// TwinCAT 3 PLC project bts_vac
// ProgramVersion: 3.1.4023.0
// libraries:
//   Tc2_Standard, * (Beckhoff Automation GmbH)
//   Tc2_System, * (Beckhoff Automation GmbH)
//   Tc2_Utilities, * (Beckhoff Automation GmbH)
//   Tc3_Module, * (Beckhoff Automation GmbH)
//   LCLS General,2.4.2,SLAC
//   LCLS Vacuum,1.4.0,SLAC - LCLS
//   LCLSVacuumSerialDriverLib,1.2.2,SLAC - LCLS
//   PMPS,0.15.3,SLAC - LCLS
// project tree:
//   DUTs/ E_TransportTube.TcDUT (not stored), ST_TransportTubeConfig.TcDUT (not stored), ST_TransportTubeDevices.TcDUT (not stored), T_TransportTube.TcDUT (not stored)
//   DUTs/Operations/ E_Op.TcDUT (not stored), E_OpStep.TcDUT (not stored)
//   DUTs/SystemStatusChecks/ E_GaugeCompOp.TcDUT (not stored)
//   DUTs/SystemStatusChecks/Switchbox/ ST_SBGaugeReadings.TcDUT, ST_SBGaugeReadingsOp.TcDUT, ST_SBPumpStatuses.TcDUT (not stored), ST_SBValveStatuses.TcDUT (not stored)
//   DUTs/SystemStatusChecks/TransportTubes/ ST_TransportTubeOps.TcDUT (not stored), ST_TransportTubeStatuses.TcDUT (not stored)
//   GVLs/ GVL_BTS_VAC.TcGVL, GVL_Constants.TcGVL (not stored), GVL_MaintainLaser.TcGVL (not stored), GVL_Operation.TcGVL (not stored), GVL_TransportTubes.TcGVL (not stored)
//   / PlcTask.TcTTO (not stored)
//   POUs/ FB_TransportTube.TcPOU (not stored), F_UpdateIO.TcPOU (not stored), MAIN.TcPOU, MaintainLaser.TcPOU (not stored), Operate.TcPOU (not stored)
//   POUs/Helpers/ F_Atm.TcPOU (not stored), F_GetTransportTube.TcPOU (not stored), F_PumpStationTurboPumpInterlock.TcPOU (not stored), F_SBVentInterlock.TcPOU (not stored)
//   POUs/Operations/Abstracts/ FB_MaintainLaserOperation.TcPOU (not stored), FB_Operation.TcPOU (not stored), FB_TTOperation.TcPOU (not stored)
//   POUs/Operations/ FB_LaserOn.TcPOU (not stored), FB_OpenTransportTube.TcPOU (not stored), FB_SlowPumpSwitchbox.TcPOU (not stored), FB_SlowVentSwitchbox.TcPOU (not stored), FB_VentTransportTube.TcPOU (not stored), FB_VentPumpStation.TcPOU (not stored), FB_PumpSwitchbox.TcPOU (not stored), FB_VentSwitchbox.TcPOU, FB_PumpTransportTube.TcPOU (not stored)
//   POUs/Operations/MaintainLaser/ FB_SwitchboxIonPumpFailure.TcPOU (not stored), FB_SwitchboxRoughingOrTurboPumpFailure.TcPOU (not stored)
//   POUs/SystemStatusChecks/ F_CompareGauge.TcPOU (not stored)
//   POUs/SystemStatusChecks/Switchbox/ F_GetSBGaugeReadings.TcPOU (not stored), F_GetSBPumpStatuses.TcPOU (not stored), F_GetSBValveStatuses.TcPOU (not stored), F_SetSBPumpStatuses.TcPOU (not stored), F_SetSBValveStatuses.TcPOU, F_VerifySBGaugeReadings.TcPOU (not stored), F_VerifySBPumpStatuses.TcPOU (not stored), F_VerifySBValveStatuses.TcPOU (not stored)
//   POUs/SystemStatusChecks/TransportTubes/ F_GetTransportTubeStatuses.TcPOU (not stored), F_SetTransportTubeStatuses.TcPOU (not stored), F_VerifyAllTransportTubeStatuses.TcPOU (not stored), F_VerifyTransportTubeStatuses.TcPOU (not stored)

// ---- DUTs/SystemStatusChecks/Switchbox/ST_SBGaugeReadings.TcDUT
(* Statuses of the gauges for the switchbox *)
TYPE ST_SBGaugeReadings :
STRUCT
	(* Gauge readings *)
	
	fDPPiraniVal : REAL; // LXLHN:GPI:03
	eDPPiraniState : E_PressureState;
	
	fDPColdCathodeVal : REAL; // LXLHN:GCC:02
	eDPColdCathodeState : E_PressureState;
	
	fPumpStationPirani1Val : REAL; // LXLHN:GPI:01
	ePumpStationPirani1State : E_PressureState;
	
	fPumpStationPirani2Val : REAL; // LXLHN:GPI:02
	ePumpStationPirani2State : E_PressureState;
	
	fPumpStationColdCathodeVal : REAL; // LXLHN:GCC:01
	ePumpStationColdCathodeState : E_PressureState;
END_STRUCT
END_TYPE

// ---- DUTs/SystemStatusChecks/Switchbox/ST_SBGaugeReadingsOp.TcDUT
(* What operations should be used to compare gauge status *)
TYPE ST_SBGaugeReadingsOp :
STRUCT
	eDPPiraniOp : E_GaugeCompOp; // LXLHN:GPI:03
	eDPColdCathodeOp : E_GaugeCompOp; // LXLHN:GCC:02
	ePumpStationPirani1Op : E_GaugeCompOp; // LXLHN:GPI:01
	ePumpStationPirani2Op : E_GaugeCompOp; // LXLHN:GPI:02
	ePumpStationColdCathodeOp : E_GaugeCompOp; // LXLHN:GCC:01
END_STRUCT
END_TYPE

// ---- GVLs/GVL_BTS_VAC.TcGVL
{attribute 'qualified_only'}
VAR_GLOBAL
	(* Valves *)	
	fb_PP_VGC_FFOut : FB_HardwareFFOutput;
	
	{attribute 'pytmc'	  :=	' pv: LXLHN:VGC:01 '}
	{attribute 'TcLinkTo' := 	'.i_xOpnLS			:=	TIIB[EL1004_02_12]^Channel 2^Input;
								 .i_xClsLS			:=	TIIB[EL1004_02_12]^Channel 1^Input;
								 .q_xOPN_DO			:=	TIIB[EL2004_02_14]^Channel 2^Output'}
	fb_PP_VGC : FB_VGC; // Gate valve, vacuum switchbox
	
	{attribute 'pytmc' 	  :=	' pv: LXLHN:VVC:01 '}
	{attribute 'TcLinkTo' := 	'.q_xOPN_DO			:=	TIIB[EL2004_02_05]^Channel 3^Output'}
	fb_PP_VVC : FB_VVC; // Turbo N2 purge
	
	
	{attribute 'pytmc'	  :=	' pv: LXLHN:VRC:01 '}
	{attribute 'TcLinkTo' := 	'.i_xOpnLS			:=	TIIB[EL1002_02_01]^Channel 2^Input;
								 .i_xClsLS			:=	TIIB[EL1002_02_01]^Channel 1^Input;
								 .q_xOPN_DO			:=	TIIB[EL2004_02_04]^Channel 1^Output'}
	fb_PP_VRC_1 : FB_VRC; // O-ring diff pump valve
	
	{attribute 'pytmc'	  :=	' pv: LXLHN:VRC:02 '}
	{attribute 'TcLinkTo' := 	'.i_xOpnLS			:=	TIIB[EL1002_02_02]^Channel 2^Input;
								 .i_xClsLS			:=	TIIB[EL1002_02_02]^Channel 1^Input;
								 .q_xOPN_DO			:=	TIIB[EL2004_02_04]^Channel 3^Output'}
	fb_PP_VRC_2 : FB_VRC; // Foreline valve
	
	{attribute 'pytmc'	  :=	' pv: LXLHN:VRC:03 '}
	{attribute 'TcLinkTo' := 	'.i_xOpnLS			:=	TIIB[EL1002_02_03]^Channel 2^Input;
								 .i_xClsLS			:=	TIIB[EL1002_02_03]^Channel 1^Input;
								 .q_xOPN_DO			:=	TIIB[EL2004_02_04]^Channel 4^Output'}
	fb_PP_VRC_3 : FB_VRC; // Slow pump valve
	
	st_VP_VVC_1 : ST_VCC_NO;
	{attribute 'pytmc' 	  :=	' pv: LXLHN:VVC:02 '}
	{attribute 'TcLinkTo' := 	'.q_xOPN_DO			:=	TIIB[EL2004_02_05]^Channel 1^Output'}
	fb_VP_VVC_1 : FB_VCC_NO; // Vent valve, Switchbox
	
	st_VP_VVC_2 : ST_VCC_NO;
	{attribute 'pytmc' 	  :=	' pv: LXLHN:VVC:032 '}
	{attribute 'TcLinkTo' := 	'.q_xOPN_DO			:=	TIIB[EL2004_02_05]^Channel 2^Output'}
	fb_VP_VVC_2 : FB_VCC_NO; // Vent valve, Slow, Switchbox

	
	(* Pumps *)
	{attribute 'pytmc' 	  := ' 	
		pv: LXLHN:PTM:01
		io: io 
	'}
	{attribute 'TcLinkTo' := 	'.i_xAtSpd			:=	TIIB[EL1004_00_03]^Channel 3^Input;
								 .i_xRemote			:=	TIIB[EL1004_00_03]^Channel 2^Input;
								 .i_xFaultNC		:=	TIIB[EL1004_00_03]^Channel 1^Output;
								 .q_RunDO			:=	TIIB[EL2004_00_04]^Channel 1^Input;
								 .q_xRemote			:=	TIIB[EL2004_00_04]^Channel 2^Input;								 
								 .q_PumpingStation	:=	TIIB[EL2004_00_04]^Channel 3^Output;'}								
	fb_PP_PTM : FB_PTM_Pfeiffer; // Turbo pump
	
	{attribute 'pytmc' 	  := ' 	
		pv: LXLHN:PMF:01
		io: io 
	'}
	{attribute 'TcLinkTo' := 	'.i_xWarning		:=	TIIB[EL1004_00_01]^Channel 4^Input;
								 .i_xAlarm			:=	TIIB[EL1004_00_01]^Channel 3^Input;
								 .i_xLocal			:=	TIIB[EL1004_00_01]^Channel 2^Output;
								 .i_xIsRun			:=	TIIB[EL1004_00_01]^Channel 1^Output;								 
								 .q_xRunDO			:=	TIIB[EL2794_00_02]^Channel 1^Input;
								 .q_xLspdDO			:=	TIIB[EL2794_00_02]^Channel 2^Input;								 
								 .q_xResetDo		:=	TIIB[EL2794_00_02]^Channel 3^Output;'}	
	fb_PP_PMF : FB_KashiyamaPump; // Roughing Pump
	
	{attribute 'pytmc'    := 	' pv: LXLHN:PP:PIP'}
	{attribute 'TcLinkTo' := 	'.i_iPRESS			:=	TIIB[EL3064_00_08]^AI Standard Channel 3^Value;
								 .i_xSP_DI			:= 	TIIB[EL1004_00_07]^Channel 3^Input;
								 .q_xHVEna_DO		:= 	TIIB[EL2794_00_06]^Channel 3^Output'}
	fb_PP_PIP : FB_PIP_Gamma; // Ion Pump, SW
	
	(* Gauges *)
	{attribute 'pytmc' 	  :=	' pv: LXLHN:GPI:01 '}
	{attribute 'TcLinkTo' := 	'.i_iPRESS_R		:=	TIIB[EL3174_01_10]^AI Standard Channel 3^Value '}
	fb_PP_GPI_1 : FB_MKS275; // Switchbox pumpline ATM gauge
	
	{attribute 'pytmc' 	  :=	' pv: LXLHN:GPI:02 '}
	{attribute 'TcLinkTo' := 	'.i_iPRESS_R		:=	TIIB[EL3174_01_11]^AI Standard Channel 1^Value '}
	fb_PP_GPI_2 : FB_MKS275; // Foreline gauge
	
	{attribute 'pytmc' 	  :=	' pv: LXLHN:GPI:03 '}
	{attribute 'TcLinkTo' := 	'.i_iPRESS_R		:=	TIIB[EL3174_01_10]^AI Standard Channel 2^Value '}
	fb_DP_GPI : FB_MKS275; // Switchbox gauge
	
	{attribute 'pytmc' 	  :=	' pv: LXLHN:GCC:01 '}
	{attribute 'TcLinkTo' := 	'.i_iPRESS_R		:=	TIIB[EL3174_01_09]^AI Standard Channel 2^Value;
								 .i_xHV_ON	    	:=	TIIB[EL1124_01_06]^Channel 1^Input;
								 .i_xDisc_Active	:=	TIIB[EL1124_01_06]^Channel 2^Input;
								 .q_xHV_DIS			:= 	TIIB[EL2624_01_02]^Channel 2^Output	'}
	fb_PP_GCC : FB_MKS500; // Switchbox pumpline Cold Cathode gauge
	
	{attribute 'pytmc' 	  :=	' pv: LXLHN:GCC:02 '}
	{attribute 'TcLinkTo' := 	'.i_iPRESS_R		:=	TIIB[EL3174_01_09]^AI Standard Channel 4^Value;
								 .i_xHV_ON	    	:=	TIIB[EL1124_01_07]^Channel 3^Input;
								 .i_xDisc_Active	:=	TIIB[EL1124_01_07]^Channel 4^Input;
								 .q_xHV_DIS			:= 	TIIB[EL2624_01_02]^Channel 4^Output	'}
	fb_DP_GCC : FB_MKS500; // Switchbox Cold Cathode gauge
	
	(* Transport Tubes *)
	// LS1
	fb_LS1_VGC_FFOut : FB_HardwareFFOutput;
	{attribute 'pytmc'	  :=	' pv: LTLHN:LS1:VGC:01 '}
	{attribute 'TcLinkTo' := 	'.i_xOpnLS			:=	TIIB[EL1004_02_06]^Channel 2^Input;
								 .i_xClsLS			:=	TIIB[EL1004_02_06]^Channel 1^Input;
								 .q_xOPN_DO			:=	TIIB[EL2004_02_08]^Channel 1^Output'}
	fb_LS1_VGC : FB_VGC; // Gate valve, Input LS1 laser Table
	{attribute 'pytmc'    := 	' pv: LTLHN:LS1:PIP:01 '}
	{attribute 'TcLinkTo' := 	'.i_iPRESS			:=	TIIB[EL3064_00_08]^AI Standard Channel 2^Value;
								 .i_xSP_DI			:= 	TIIB[EL1004_00_07]^Channel 2^Input;
								 .q_xHVEna_DO		:= 	TIIB[EL2794_00_06]^Channel 2^Output'}
	fb_LS1_PIP : FB_PIP_Gamma; // Ion Pump, input tube LS1
	{attribute 'pytmc' 	  :=	' pv: LTLHN:LS1:GPI:01 '}
	{attribute 'TcLinkTo' := 	'.i_iPRESS_R		:=	TIIB[EL3174_01_10]^AI Standard Channel 4^Value '}
	fb_LS1_GPI : FB_MKS275; // Input tube LS1 ATM gauge
	{attribute 'pytmc' 	  :=	' pv: LTLHN:LS1:GCC:01 '}
	{attribute 'TcLinkTo' := 	'.i_iPRESS_R		:=	TIIB[EL3174_01_09]^AI Standard Channel 3^Value;
								 .i_xHV_ON	    	:=	TIIB[EL1124_01_06]^Channel 3^Input;
								 .i_xDisc_Active	:=	TIIB[EL1124_01_06]^Channel 4^Input;
								 .q_xHV_DIS			:= 	TIIB[EL2624_01_02]^Channel 3^Output	'}
	fb_LS1_GCC : FB_MKS500; // Input tube LS1, Cold Cathode gauge
	
	// LS5
	fb_LS5_VGC_FFOut : FB_HardwareFFOutput;
	{attribute 'pytmc'	  :=	' pv: LTLHN:LS5:VGC:01 '}
	{attribute 'TcLinkTo' := 	'.i_xOpnLS			:=	TIIB[EL1004_02_09]^Channel 4^Input;
								 .i_xClsLS			:=	TIIB[EL1004_02_09]^Channel 3^Input;
								 .q_xOPN_DO			:=	TIIB[EL2004_02_11]^Channel 2^Output'}
	fb_LS5_VGC : FB_VGC; // Gate valve, Input LS5 laser Table
	{attribute 'pytmc'    := 	' pv: LTLHN:LS5:PIP:01 '}
	{attribute 'TcLinkTo' := 	'.i_iPRESS			:=	TIIB[EL3064_00_11]^AI Standard Channel 4^Value;
								 .i_xSP_DI			:= 	TIIB[EL1004_00_10]^Channel 4^Input;
								 .q_xHVEna_DO		:= 	TIIB[EL2794_00_09]^Channel 4^Output'}
	fb_LS5_PIP : FB_PIP_Gamma; // Ion Pump, input tube LS5
	{attribute 'pytmc' 	  :=	' pv: LTLHN:LS5:GPI:01 '}
	{attribute 'TcLinkTo' := 	'.i_iPRESS_R		:=	TIIB[EL3174_03_13]^AI Standard Channel 1^Value '}
	fb_LS5_GPI : FB_MKS275; // Input tube LS5 ATM gauge
	{attribute 'pytmc' 	  :=	' pv: LTLHN:LS5:GCC:01 '}
	{attribute 'TcLinkTo' := 	'.i_iPRESS_R		:=	TIIB[EL3174_03_11]^AI Standard Channel 1^Value;
								 .i_xHV_ON	    	:=	TIIB[EL1124_03_08]^Channel 1^Input;
								 .i_xDisc_Active	:=	TIIB[EL1124_03_08]^Channel 2^Input;
								 .q_xHV_DIS			:= 	TIIB[EL2624_03_02]^Channel 1^Output	'}
	fb_LS5_GCC : FB_MKS500; // Input tube LS5, Cold Cathode gauge
	
	// LS8
	fb_LS8_VGC_FFOut : FB_HardwareFFOutput;
	{attribute 'pytmc'	  :=	' pv: LTLHN:LS8:VGC:01 '}
	{attribute 'TcLinkTo' := 	'.i_xOpnLS			:=	TIIB[EL1004_02_09]^Channel 2^Input;
								 .i_xClsLS			:=	TIIB[EL1004_02_09]^Channel 1^Input;
								 .q_xOPN_DO			:=	TIIB[EL2004_02_11]^Channel 3^Output'}
	fb_LS8_VGC : FB_VGC; // Gate valve, Input LS8 laser Table
	{attribute 'pytmc'    := 	' pv: LTLHN:LS8:PIP:01 '}
	{attribute 'TcLinkTo' := 	'.i_iPRESS			:=	TIIB[EL3064_00_11]^AI Standard Channel 3^Value;
								 .i_xSP_DI			:= 	TIIB[EL1004_00_10]^Channel 3^Input;
								 .q_xHVEna_DO		:= 	TIIB[EL2794_00_09]^Channel 3^Output'}
	fb_LS8_PIP : FB_PIP_Gamma; // Ion Pump, input tube LS8
	{attribute 'pytmc' 	  :=	' pv: LTLHN:LS8:GPI:01 '}
	{attribute 'TcLinkTo' := 	'.i_iPRESS_R		:=	TIIB[EL3174_03_13]^AI Standard Channel 2^Value '}
	fb_LS8_GPI : FB_MKS275; // Input tube LS8 ATM gauge
	{attribute 'pytmc' 	  :=	' pv: LTLHN:LS8:GCC:01 '}
	{attribute 'TcLinkTo' := 	'.i_iPRESS_R		:=	TIIB[EL3174_03_11]^AI Standard Channel 2^Value;
								 .i_xHV_ON	    	:=	TIIB[EL1124_03_08]^Channel 3^Input;
								 .i_xDisc_Active	:=	TIIB[EL1124_03_08]^Channel 4^Input;
								 .q_xHV_DIS			:= 	TIIB[EL2624_03_02]^Channel 2^Output	'}
	fb_LS8_GCC : FB_MKS500; // Input tube LS8, Cold Cathode gauge

	// LD2
	fb_LD2_VGC_FFOut : FB_HardwareFFOutput;
	{attribute 'pytmc'	  :=	' pv: LTLHN:LD2:VGC:01 '}
	{attribute 'TcLinkTo' := 	'.i_xOpnLS			:=	TIIB[EL1004_02_12]^Channel 4^Input;
								 .i_xClsLS			:=	TIIB[EL1004_02_12]^Channel 3^Input;
								 .q_xOPN_DO			:=	TIIB[EL2004_02_14]^Channel 3^Output'}
	fb_LD2_VGC : FB_VGC; // Gate valve, Output tube LD2 laser Table
	{attribute 'pytmc'    := 	' pv: LTLHN:LD2:PIP:01 '}
	{attribute 'TcLinkTo' := 	'.i_iPRESS			:=	TIIB[EL3064_00_08]^AI Standard Channel 1^Value;
								 .i_xSP_DI			:= 	TIIB[EL1004_00_07]^Channel 1^Input;
								 .q_xHVEna_DO		:= 	TIIB[EL2794_00_06]^Channel 1^Output'}
	fb_LD2_PIP : FB_PIP_Gamma; // Ion Pump, output tube LD2
	{attribute 'pytmc' 	  :=	' pv: LTLHN:LD2:GPI:01 '}
	{attribute 'TcLinkTo' := 	'.i_iPRESS_R		:=	TIIB[EL3174_01_10]^AI Standard Channel 1^Value '}
	fb_LD2_GPI : FB_MKS275; // Output tube LD2 ATM gauge
	{attribute 'pytmc' 	  :=	' pv: LTLHN:LD2:GCC:01 '}
	{attribute 'TcLinkTo' := 	'.i_iPRESS_R		:=	TIIB[EL3174_01_09]^AI Standard Channel 1^Value;
								 .i_xHV_ON	    	:=	TIIB[EL1124_01_07]^Channel 1^Input;
								 .i_xDisc_Active	:=	TIIB[EL1124_01_07]^Channel 2^Input;
								 .q_xHV_DIS			:= 	TIIB[EL2624_01_02]^Channel 1^Output	'}
	fb_LD2_GCC : FB_MKS500; // Output tube LD2, Cold Cathode gauge
	
	// LD4
	fb_LD4_VGC_FFOut : FB_HardwareFFOutput;
	{attribute 'pytmc'	  :=	' pv: LTLHN:LD4:VGC:01 '}
	{attribute 'TcLinkTo' := 	'.i_xOpnLS			:=	TIIB[EL1004_02_10]^Channel 2^Input;
								 .i_xClsLS			:=	TIIB[EL1004_02_10]^Channel 1^Input;
								 .q_xOPN_DO			:=	TIIB[EL2004_02_11]^Channel 1^Output'}
	fb_LD4_VGC : FB_VGC; // Gate valve, Output tube LD4 laser Table
	{attribute 'pytmc'    := 	' pv: LTLHN:LD4:PIP:01 '}
	{attribute 'TcLinkTo' := 	'.i_iPRESS			:=	TIIB[EL3064_00_11]^AI Standard Channel 1^Value;
								 .i_xSP_DI			:= 	TIIB[EL1004_00_10]^Channel 1^Input;
								 .q_xHVEna_DO		:= 	TIIB[EL2794_00_09]^Channel 1^Output'}
	fb_LD4_PIP : FB_PIP_Gamma; // Ion Pump, output tube LD4
	{attribute 'pytmc' 	  :=	' pv: LTLHN:LD4:GPI:01 '}
	{attribute 'TcLinkTo' := 	'.i_iPRESS_R		:=	TIIB[EL3174_03_13]^AI Standard Channel 4^Value '}
	fb_LD4_GPI : FB_MKS275; // Output tube LD4 ATM gauge
	{attribute 'pytmc' 	  :=	' pv: LTLHN:LD4:GCC:01 '}
	{attribute 'TcLinkTo' := 	'.i_iPRESS_R		:=	TIIB[EL3174_03_11]^AI Standard Channel 4^Value;
								 .i_xHV_ON	    	:=	TIIB[EL1124_03_09]^Channel 3^Input;
								 .i_xDisc_Active	:=	TIIB[EL1124_03_09]^Channel 4^Input;
								 .q_xHV_DIS			:= 	TIIB[EL2624_03_02]^Channel 4^Output	'}
	fb_LD4_GCC : FB_MKS500; // Output tube LD4, Cold Cathode gauge
	
	// LD6
	fb_LD6_VGC_FFOut : FB_HardwareFFOutput;
	{attribute 'pytmc'	  :=	' pv: LTLHN:LD6:VGC:01 '}
	{attribute 'TcLinkTo' := 	'.i_xOpnLS			:=	TIIB[EL1004_02_13]^Channel 4^Input;
								 .i_xClsLS			:=	TIIB[EL1004_02_13]^Channel 3^Input;
								 .q_xOPN_DO			:=	TIIB[EL2004_02_14]^Channel 4^Output'}
	fb_LD6_VGC : FB_VGC; // Gate valve, Output tube LD6 laser Table
	{attribute 'pytmc'    := 	' pv: LTLHN:LD6:PIP:01 '}
	{attribute 'TcLinkTo' := 	'.i_iPRESS			:=	TIIB[EL3064_00_11]^AI Standard Channel 2^Value;
								 .i_xSP_DI			:= 	TIIB[EL1004_00_10]^Channel 2^Input;
								 .q_xHVEna_DO		:= 	TIIB[EL2794_00_09]^Channel 2^Output'}
	fb_LD6_PIP : FB_PIP_Gamma; // Ion Pump, output tube LD6
	{attribute 'pytmc' 	  :=	' pv: LTLHN:LD6:GPI:01 '}
	{attribute 'TcLinkTo' := 	'.i_iPRESS_R		:=	TIIB[EL3174_03_13]^AI Standard Channel 3^Value '}
	fb_LD6_GPI : FB_MKS275; // Output tube LD6 ATM gauge
	{attribute 'pytmc' 	  :=	' pv: LTLHN:LD6:GCC:01 '}
	{attribute 'TcLinkTo' := 	'.i_iPRESS_R		:=	TIIB[EL3174_03_11]^AI Standard Channel 3^Value;
								 .i_xHV_ON	    	:=	TIIB[EL1124_03_09]^Channel 1^Input;
								 .i_xDisc_Active	:=	TIIB[EL1124_03_09]^Channel 2^Input;
								 .q_xHV_DIS			:= 	TIIB[EL2624_03_02]^Channel 3^Output	'}
	fb_LD6_GCC : FB_MKS500; // Output tube LD6, Cold Cathode gauge

	// LD8
	fb_LD8_VGC_FFOut : FB_HardwareFFOutput;
	{attribute 'pytmc'	  :=	' pv: LTLHN:LD8:VGC:01 '}
	{attribute 'TcLinkTo' := 	'.i_xOpnLS			:=	TIIB[EL1004_02_07]^Channel 4^Input;
								 .i_xClsLS			:=	TIIB[EL1004_02_07]^Channel 3^Input;
								 .q_xOPN_DO			:=	TIIB[EL2004_02_07]^Channel 4^Output'}
	fb_LD8_VGC : FB_VGC; // Gate valve, Output tube LD8 laser Table
	{attribute 'pytmc'    := 	' pv: LTLHN:LD8:PIP:01 '}
	{attribute 'TcLinkTo' := 	'.i_iPRESS			:=	TIIB[EL3064_00_08]^AI Standard Channel 4^Value;
								 .i_xSP_DI			:= 	TIIB[EL1004_00_07]^Channel 4^Input;
								 .q_xHVEna_DO		:= 	TIIB[EL2794_00_06]^Channel 4^Output'}
	fb_LD8_PIP : FB_PIP_Gamma; // Ion Pump, output tube LD8
	{attribute 'pytmc' 	  :=	' pv: LTLHN:LD8:GPI:01 '}
	{attribute 'TcLinkTo' := 	'.i_iPRESS_R		:=	TIIB[EL3174_01_11]^AI Standard Channel 2^Value '}
	fb_LD8_GPI : FB_MKS275; // Output tube LD8 ATM gauge
	{attribute 'pytmc' 	  :=	' pv: LTLHN:LD8:GCC:01 '}
	{attribute 'TcLinkTo' := 	'.i_iPRESS_R		:=	TIIB[EL3174_01_11]^AI Standard Channel 3^Value;
								 .i_xHV_ON	    	:=	TIIB[EL1124_01_08]^Channel 1^Input;
								 .i_xDisc_Active	:=	TIIB[EL1124_01_08]^Channel 2^Input;
								 .q_xHV_DIS			:= 	TIIB[EL2624_01_01]^Channel 4^Output	'}
	fb_LD8_GCC : FB_MKS500; // Output tube LD8, Cold Cathode gauge
	
	// LD9
	fb_LD9_VGC_FFOut : FB_HardwareFFOutput;
	{attribute 'pytmc'	  :=	' pv: LTLHN:LD9:VGC:01 '}
	{attribute 'TcLinkTo' := 	'.i_xOpnLS			:=	TIIB[EL1004_02_06]^Channel 4^Input;
								 .i_xClsLS			:=	TIIB[EL1004_02_06]^Channel 3^Input;
								 .q_xOPN_DO			:=	TIIB[EL2004_02_08]^Channel 2^Output'}
	fb_LD9_VGC : FB_VGC; // Gate valve, Output tube LD9 laser Table
	{attribute 'pytmc'    := 	' pv: LTLHN:LD9:PIP:01 '}
	{attribute 'TcLinkTo' := 	'.i_iPRESS			:=	TIIB[EL3064_00_14]^AI Standard Channel 2^Value;
								 .i_xSP_DI			:= 	TIIB[EL1004_00_13]^Channel 2^Input;
								 .q_xHVEna_DO		:= 	TIIB[EL2794_00_12]^Channel 2^Output'}
	fb_LD9_PIP : FB_PIP_Gamma; // Ion Pump, output tube LD9
	{attribute 'pytmc' 	  :=	' pv: LTLHN:LD9:GPI:01 '}
	{attribute 'TcLinkTo' := 	'.i_iPRESS_R		:=	TIIB[EL3174_03_12]^AI Standard Channel 1^Value '}
	fb_LD9_GPI : FB_MKS275; // Output tube LD9 ATM gauge
	{attribute 'pytmc' 	  :=	' pv: LTLHN:LD9:GCC:01 '}
	{attribute 'TcLinkTo' := 	'.i_iPRESS_R		:=	TIIB[EL3174_03_10]^AI Standard Channel 1^Value;
								 .i_xHV_ON	    	:=	TIIB[EL1124_03_06]^Channel 1^Input;
								 .i_xDisc_Active	:=	TIIB[EL1124_03_06]^Channel 2^Input;
								 .q_xHV_DIS			:= 	TIIB[EL2624_03_01]^Channel 1^Output	'}
	fb_LD9_GCC : FB_MKS500; // Output tube LD9, Cold Cathode gauge

	// LD10
	fb_LD10_VGC_FFOut : FB_HardwareFFOutput;
	{attribute 'pytmc'	  :=	' pv: LTLHN:LD10:VGC:01 '}
	{attribute 'TcLinkTo' := 	'.i_xOpnLS			:=	TIIB[EL1004_02_07]^Channel 2^Input;
								 .i_xClsLS			:=	TIIB[EL1004_02_07]^Channel 1^Input;
								 .q_xOPN_DO			:=	TIIB[EL2004_02_07]^Channel 3^Output'}
	fb_LD10_VGC : FB_VGC; // Gate valve, Output tube LD10 laser Table
	{attribute 'pytmc'    := 	' pv: LTLHN:LD10:PIP:01 '}
	{attribute 'TcLinkTo' := 	'.i_iPRESS			:=	TIIB[EL3064_00_14]^AI Standard Channel 1^Value;
								 .i_xSP_DI			:= 	TIIB[EL1004_00_13]^Channel 1^Input;
								 .q_xHVEna_DO		:= 	TIIB[EL2794_00_12]^Channel 1^Output'}
	fb_LD10_PIP : FB_PIP_Gamma; // Ion Pump, output tube LD10
	{attribute 'pytmc' 	  :=	' pv: LTLHN:LD10:GPI:01 '}
	{attribute 'TcLinkTo' := 	'.i_iPRESS_R		:=	TIIB[EL3174_03_12]^AI Standard Channel 2^Value '}
	fb_LD10_GPI : FB_MKS275; // Output tube LD10 ATM gauge
	{attribute 'pytmc' 	  :=	' pv: LTLHN:LD10:GCC:01 '}
	{attribute 'TcLinkTo' := 	'.i_iPRESS_R		:=	TIIB[EL3174_03_10]^AI Standard Channel 2^Value;
								 .i_xHV_ON	    	:=	TIIB[EL1124_03_07]^Channel 3^Input;
								 .i_xDisc_Active	:=	TIIB[EL1124_03_07]^Channel 4^Input;
								 .q_xHV_DIS			:= 	TIIB[EL2624_03_01]^Channel 2^Output	'}
	fb_LD10_GCC : FB_MKS500; // Output tube LD10, Cold Cathode gauge	
	
	// LD14
	fb_LD14_VGC_FFOut : FB_HardwareFFOutput;
	{attribute 'pytmc'	  :=	' pv: LTLHN:LD14:VGC:01 '}
	{attribute 'TcLinkTo' := 	'.i_xOpnLS			:=	TIIB[EL1004_02_10]^Channel 4^Input;
								 .i_xClsLS			:=	TIIB[EL1004_02_10]^Channel 3^Input;
								 .q_xOPN_DO			:=	TIIB[EL2004_02_11]^Channel 4^Output'}
	fb_LD14_VGC : FB_VGC; // Gate valve, Output tube LD14 laser Table
	{attribute 'pytmc'    := 	' pv: LTLHN:LD14:PIP:01 '}
	{attribute 'TcLinkTo' := 	'.i_iPRESS			:=	TIIB[EL3064_00_14]^AI Standard Channel 3^Value;
								 .i_xSP_DI			:= 	TIIB[EL1004_00_13]^Channel 3^Input;
								 .q_xHVEna_DO		:= 	TIIB[EL2794_00_12]^Channel 3^Output'}
	fb_LD14_PIP : FB_PIP_Gamma; // Ion Pump, output tube LD14
	{attribute 'pytmc' 	  :=	' pv: LTLHN:LD14:GPI:01 '}
	{attribute 'TcLinkTo' := 	'.i_iPRESS_R		:=	TIIB[EL3174_03_12]^AI Standard Channel 3^Value '}
	fb_LD14_GPI : FB_MKS275; // Output tube LD14 ATM gauge
	{attribute 'pytmc' 	  :=	' pv: LTLHN:LD14:GCC:01 '}
	{attribute 'TcLinkTo' := 	'.i_iPRESS_R		:=	TIIB[EL3174_03_10]^AI Standard Channel 3^Value;
								 .i_xHV_ON	    	:=	TIIB[EL1124_03_07]^Channel 1^Input;
								 .i_xDisc_Active	:=	TIIB[EL1124_03_07]^Channel 2^Input;
								 .q_xHV_DIS			:= 	TIIB[EL2624_03_01]^Channel 3^Output	'}
	fb_LD14_GCC : FB_MKS500; // Output tube LD14, Cold Cathode gauge

END_VAR

// ---- POUs/MAIN.TcPOU
PROGRAM MAIN
VAR
END_VAR

(* Update physical IO signals *)
F_UpdateIO();

(* Update transport tubes *)
GVL_TransportTubes.fbLS1(
	i_stConfig := GVL_TransportTubes.stLS1, 
	i_bLaserExtIntl := TRUE
);

GVL_TransportTubes.fbLS5(
	i_stConfig := GVL_TransportTubes.stLS5, 
	i_bLaserExtIntl := TRUE
);

GVL_TransportTubes.fbLS8(
	i_stConfig := GVL_TransportTubes.stLS8, 
	i_bLaserExtIntl := TRUE
);

GVL_TransportTubes.fbLD2(
	i_stConfig := GVL_TransportTubes.stLD2,
	i_bLaserExtIntl := TRUE
);

GVL_TransportTubes.fbLD4(
	i_stConfig := GVL_TransportTubes.stLD4,
	i_bLaserExtIntl := TRUE
);

GVL_TransportTubes.fbLD6(
	i_stConfig := GVL_TransportTubes.stLD6,
	i_bLaserExtIntl := TRUE
);

GVL_TransportTubes.fbLD14(
	i_stConfig := GVL_TransportTubes.stLD14,
	i_bLaserExtIntl := TRUE
);

GVL_TransportTubes.fbLD10(
	i_stConfig := GVL_TransportTubes.stLD10,
	i_bLaserExtIntl := TRUE
);

GVL_TransportTubes.fbLD9(
	i_stConfig := GVL_TransportTubes.stLD9,
	i_bLaserExtIntl := TRUE
);

GVL_TransportTubes.fbLD8(
	i_stConfig := GVL_TransportTubes.stLD8,
	i_bLaserExtIntl := TRUE
);

END_PROGRAM

// ---- POUs/Operations/FB_VentSwitchbox.TcPOU
(* Operation for venting the switchbox *)
FUNCTION_BLOCK FB_VentSwitchbox EXTENDS FB_Operation
VAR_STAT CONSTANT
	(* Expected system states before operation starts*)
	stExpPumpStatus : ST_SBPumpStatuses := (
		bRoughingPumpOn:= TRUE, 
		bTurboPumpOn:= FALSE, 
		bIonPumpOn:= TRUE);
	
	stExpValveStatus : ST_SBValveStatuses := (
		bGateValveOpen:= TRUE, 
		bVentValveOpen:= FALSE, 
		bORingPumpValveOpen:= TRUE, 
		bForelineValveOpen:= TRUE,
		bSlowPumpValveOpen:= FALSE,
		bSBVentOpen:= FALSE,  
		bSBSlowVentOpen:= FALSE);
	
	stExpGaugeReadings : ST_SBGaugeReadings := (
		eDPPiraniState:= E_PressureState.ValidLo,
		fDPColdCathodeVal:= 1E-5,
		ePumpStationPirani1State:= E_PressureState.ValidLo,
		ePumpStationPirani2State:= E_PressureState.ValidLo,
		fPumpStationColdCathodeVal:= 1E-5
	);
	stGaugeReadingsOp : ST_SBGaugeReadingsOp := (
		eDPPiraniOp:= E_GaugeCompOp.STATE, 
		eDPColdCathodeOp:= E_GaugeCompOp._LTE, 
		ePumpStationPirani1Op:= E_GaugeCompOp.STATE, 
		ePumpStationPirani2Op:= E_GaugeCompOp.STATE, 
		ePumpStationColdCathodeOp:= E_GaugeCompOp._LTE);
		
	stExpTTStatus : ST_TransportTubeStatuses := (bGateValveOpen:= FALSE);
	stTTOp : ST_TransportTubeOps := (bIonPumpIgnore:= TRUE);
		
	(* Expected system states after operation finishes *)
	stFinExpPumpStatus : ST_SBPumpStatuses := (
		bRoughingPumpOn:= FALSE, 
		bTurboPumpOn:= FALSE, 
		bIonPumpOn:= FALSE);
	
	stFinExpValveStatus : ST_SBValveStatuses := (
		bGateValveOpen:= FALSE, 
		bVentValveOpen:= FALSE, 
		bORingPumpValveOpen:= FALSE, 
		bForelineValveOpen:= FALSE, 
		bSlowPumpValveOpen:= FALSE,
		bSBVentOpen:= FALSE,  
		bSBSlowVentOpen:= FALSE);
	
	stFinExpGaugeReadings : ST_SBGaugeReadings := (
		eDPColdCathodeState := E_PressureState.Off,
		ePumpStationColdCathodeState := E_PressureState.Off
	);
	stFinGaugeReadingsOp : ST_SBGaugeReadingsOp := (
		eDPPiraniOp:= E_GaugeCompOp.ATM, 
		eDPColdCathodeOp:= E_GaugeCompOp.STATE, 
		ePumpStationPirani1Op:= E_GaugeCompOp.ATM, 
		ePumpStationPirani2Op:= E_GaugeCompOp.ATM, 
		ePumpStationColdCathodeOp:= E_GaugeCompOp.STATE);
		
	stFinExpTTStatus : ST_TransportTubeStatuses := (bGateValveOpen:= FALSE);
	stFinTTOp : ST_TransportTubeOps := (bIonPumpIgnore:= TRUE);
		
	(* Timeout constants *)
	VENT_TIMEOUT : TIME := T#20M;
END_VAR

SUPER^(iq_sMessageBuffer := iq_sMessageBuffer);

CASE eStep OF
E_OpStep.IDLE: // Do nothing

E_OpStep.START: // Verify system status
	M_RunTimeoutTimer(STATUS_CHECK_TIMEOUT);
	M_SetMessage('Verifying system status');
	
	IF F_VerifySBPumpStatuses(stExpStatus := stExpPumpStatus, bEnforce := TRUE)
		AND F_VerifySBValveStatuses(stExpStatus := stExpValveStatus, bEnforce := TRUE)
		AND F_VerifySBGaugeReadings(stExpReadings := stExpGaugeReadings, stReadingsOp := stGaugeReadingsOp)
		AND F_VerifyAllTransportTubeStatuses(stExpStatus := stExpTTStatus, 
			stStatusOp := stTTOp,
			bEnforce := TRUE)
	THEN // System status check 
		M_ResetTimeoutTimer();
		M_SetMessage('Closing gate valve');
		eStep := E_OpStep.VSB_CLOSE_GATE_VALVE;
	END_IF
	
E_OpStep.VSB_CLOSE_GATE_VALVE:
	M_RunTimeoutTimer(VALVE_TIMEOUT);
	
	// Close gate valve to pump station to isolate pumps
	GVL_BTS_VAC.fb_PP_VGC.M_Set_OPN_SW(FALSE);
	
	IF GVL_BTS_VAC.fb_PP_VGC.M_IsClosed() THEN
		M_ResetTimeoutTimer();
		M_SetMessage('Closing foreline valve');
		eStep := E_OpStep.VSB_CLOSE_FORELINE_VALVE;
	END_IF
	
E_OpStep.VSB_CLOSE_FORELINE_VALVE:
	M_RunTimeoutTimer(VALVE_TIMEOUT);
	
	// Close valves to pumping station to isolate pumps
	GVL_BTS_VAC.fb_PP_VRC_2.M_Set_OPN_SW(FALSE);
	
	IF GVL_BTS_VAC.fb_PP_VRC_2.iq_stValve.eState = E_ValvePositionState.CLOSED THEN
		M_ResetTimeoutTimer();
		M_SetMessage('Turning off roughing and ion pump');
		eStep := E_OpStep.VSB_TURN_OFF_PUMPS;
	END_IF
	
E_OpStep.VSB_TURN_OFF_PUMPS:
	M_RunTimeoutTimer(PUMP_TIMEOUT);
	
	// Turn off pumping station pumps
	GVL_BTS_VAC.fb_PP_PMF.M_Run(FALSE);
	GVL_BTS_VAC.fb_PP_PIP.M_Run(FALSE);
	
	IF GVL_BTS_VAC.fb_PP_PMF.q_stPump.eState = E_PumpState.pumpSTOPPED AND NOT GVL_BTS_VAC.fb_PP_PIP.i_xSP_DI THEN
		M_ResetTimeoutTimer();
		M_SetMessage('Closing O-Ring valve');
		eStep := E_OpStep.VSB_CLOSE_ORING_VALVE;
	END_IF
	
E_OpStep.VSB_CLOSE_ORING_VALVE:
	M_RunTimeoutTimer(VALVE_TIMEOUT);
	
	// Close O-Ring pump valve
	GVL_BTS_VAC.fb_PP_VRC_1.M_Set_OPN_SW(FALSE);

	IF GVL_BTS_VAC.fb_PP_VRC_1.iq_stValve.eState = E_ValvePositionState.CLOSED THEN
		M_ResetTimeoutTimer();
		M_SetMessage('Venting');
		eStep := E_OpStep.VSB_VENT;
	END_IF
	
E_OpStep.VSB_VENT:
	M_RunTimeoutTimer(VENT_TIMEOUT);
		
	// Open switchbox vent
	GVL_BTS_VAC.fb_VP_VVC_1.M_Open(TRUE);
	
	// Vent until atmospheric pressure reached in the switchbox
	IF F_Atm(GVL_BTS_VAC.fb_DP_GPI.PG.rPRESS) THEN
		M_ResetTimeoutTimer();
		eStep := E_OpStep.VSB_CLOSE_VENT;
	END_IF
	

E_OpStep.VSB_CLOSE_VENT:
	GVL_BTS_VAC.fb_VP_VVC_1.M_Open(FALSE);
	// How to verfiy the vent is closed?
	eStep := E_OpStep.VSB_FINISH;
	
E_OpStep.VSB_FINISH:
	IF F_VerifySBPumpStatuses(stExpStatus := stFinExpPumpStatus, bEnforce := FALSE)
		AND F_VerifySBValveStatuses(stExpStatus := stFinExpValveStatus, bEnforce := FALSE)
		AND F_VerifySBGaugeReadings(stExpReadings := stFinExpGaugeReadings, stReadingsOp := stFinGaugeReadingsOp)
		AND F_VerifyAllTransportTubeStatuses(stExpStatus := stFinExpTTStatus, 
			stStatusOp := stFinTTOp,
			bEnforce := FALSE)
	THEN
		M_Finish();
	ELSE
		M_FatalError('End system status check failed');
	END_IF
	
ELSE
	M_FatalError('Operation is in invalid state');
END_CASE

END_FUNCTION_BLOCK

// ---- POUs/SystemStatusChecks/Switchbox/F_SetSBValveStatuses.TcPOU
FUNCTION F_SetSBValveStatuses : BOOL
VAR_INPUT
	stExpStatuses : ST_SBValveStatuses;
END_VAR
VAR
END_VAR

GVL_BTS_VAC.fb_PP_VGC.M_Set_OPN_SW(stExpStatuses.bGateValveOpen);
GVL_BTS_VAC.fb_PP_VVC.M_Open(stExpStatuses.bVentValveOpen);
GVL_BTS_VAC.fb_PP_VRC_1.M_Set_OPN_SW(stExpStatuses.bORingPumpValveOpen); 
GVL_BTS_VAC.fb_PP_VRC_2.M_Set_OPN_SW(stExpStatuses.bForelineValveOpen);
GVL_BTS_VAC.fb_PP_VRC_3.M_Set_OPN_SW(stExpStatuses.bSBSlowVentOpen);
GVL_BTS_VAC.fb_VP_VVC_1.M_Open(stExpStatuses.bSBVentOpen);
GVL_BTS_VAC.fb_VP_VVC_2.M_Open(stExpStatuses.bSBSlowVentOpen);

END_FUNCTION
